PROGRAM SEQ_COSMO
VAR_INPUT
	COSMO_sequence	: UINT;
END_VAR

VAR
	process_V	: UINT; //COSMO to Pitstop
	process_W	: UINT; //COSMO to Reject Out
	process_X	: UINT; //Conveyor to Pitstop
	process_G	: UINT; //KR1 GET Magnet	
END_VAR


IF NOT AUTO_MODE.COSMO_LOAD OR GVL.KR1_EOAT_SUCTION OR GVL.LAYERPAD OR AUTO_MODE.FG_PACKING THEN
	RETURN;
END_IF

CASE COSMO_sequence OF
	0:
		process_V	:= 0;
		process_W	:= 0;
		process_X	:= 0;
		process_G	:= 0;
		COSMO_sequence := 1;		
		GVL.COSMO_UNLOAD := TRUE;
		AUTO_MODE.processnameCOSMO := CONCAT(MSG.COMP_CM,MSG.ACTION_INIT);
		LOGPROCESS( spLogComp	 := MSG.COMP_CM, 
		 			spLogAction	 := MSG.ACTION_INIT, 
		 			spLogStatus	 := MSG.STATUS_DONE,
	 	 		 	plogFlag	 := TRUE);
		
	// Get Magnet -------------------------------------------------------------------------------------------------------------	
	1:
		IF NOT GVL.KR1_EOAT_FILL AND NOT GVL.KR1_EOAT_SUCTION THEN
			IF process_G = 0 THEN
				IF KR1.Idle THEN
//					KR1.PLC_O_D3.0 := TRUE; //200
					KR1.bOutBit[3,0] := TRUE;
					AUTO_MODE.processnameCOSMO := CONCAT(MSG.COMP_CM,MSG.ACTION_GET_MAGNET);
					AUTO_MODE.processnameCOSMO := CONCAT(AUTO_MODE.processnameCOSMO,MSG.STATUS_RUN);
					LOGPROCESS( spLogComp	 := MSG.COMP_CM, 
								spLogAction	 := MSG.ACTION_GET_MAGNET, 
								spLogStatus	 := MSG.STATUS_RUN,
								plogFlag	 := TRUE);
					process_G := 1;
					RETURN;
				END_IF
			ELSIF process_G = 1 THEN
//				KR1.PLC_O_D3.0 := TRUE; //200
				KR1.bOutBit[3,0] := TRUE;
				IF NOT KR1.bInBit[3,0] THEN
//					KR1.PLC_O_D3.0 := FALSE; //200	
					KR1.bOutBit[3,0] := FALSE;
					AUTO_MODE.processnameCOSMO := CONCAT(MSG.COMP_CM,MSG.ACTION_GET_MAGNET);
					AUTO_MODE.processnameCOSMO := CONCAT(AUTO_MODE.processnameCOSMO,MSG.STATUS_ACK);
					LOGPROCESS( spLogComp	 := MSG.COMP_CM, 
								spLogAction	 := MSG.ACTION_GET_MAGNET, 
								spLogStatus	 := MSG.STATUS_ACK,
								plogFlag	 := TRUE);
					process_G := 2;
					RETURN;
				END_IF	
			ELSIF process_G = 2 THEN
//				KR1.PLC_O_D3.0 := FALSE; //200
				KR1.bOutBit[3,0] := FALSE;	
				IF KR1.bInBit[3,0] THEN
					AUTO_MODE.processnameCOSMO := CONCAT(MSG.COMP_CM,MSG.ACTION_GET_MAGNET);
					AUTO_MODE.processnameCOSMO := CONCAT(AUTO_MODE.processnameCOSMO,MSG.STATUS_DONE);
					LOGPROCESS( spLogComp	 := MSG.COMP_CM, 
								spLogAction	 := MSG.ACTION_GET_MAGNET, 
								spLogStatus	 := MSG.STATUS_DONE,
								plogFlag	 := TRUE);
					process_G:= 3;
					RETURN;
				END_IF	
			ELSIF process_G = 3 THEN
				IF KR1.Idle THEN
					AUTO_MODE.processnameCOSMO := CONCAT(MSG.COMP_CM,MSG.ACTION_GET_MAGNET);
					AUTO_MODE.processnameCOSMO := CONCAT(AUTO_MODE.processnameCOSMO,MSG.STATUS_COMP);
					LOGPROCESS( spLogComp	 := MSG.COMP_CM, 
								spLogAction	 := MSG.ACTION_GET_MAGNET, 
								spLogStatus	 := MSG.STATUS_COMP,
								plogFlag	 := TRUE);
					process_G := 4;
					COSMO_sequence := 2;
					AUTO_MODE.next_step := FALSE;
					GVL.KR1_EOAT_FILL := TRUE;
				END_IF
			END_IF
		ELSE
			COSMO_sequence := 2;
		END_IF
		
	// COSMO test --------------------------------------------------------------------------------------------------------------		
	2: 
		IF GVL.COSMO_OK THEN
			GVL.COSMO_Run := FALSE;
			AUTO_MODE.COSMO_RUN := FALSE;
			AUTO_MODE.processnameCOSMO := CONCAT(MSG.COMP_CM,MSG.ACTION_COSMO_PASS);
			AUTO_MODE.processnameCOSMO := CONCAT(AUTO_MODE.processnameCOSMO,MSG.STATUS_DONE);
			LOGPROCESS( spLogComp	 := MSG.COMP_CM, 
						spLogAction	 := MSG.ACTION_COSMO_PASS, 
						spLogStatus	 := MSG.STATUS_DONE,
						plogFlag	 := TRUE);
			COSMO_sequence := 3;
			AUTO_MODE.next_step := FALSE;
			AUTO_MODE.CLEAR_COSMO := TRUE;
			RETURN;
		ELSIF GVL.COSMO_NOTOK THEN
			GVL.COSMO_Run := FALSE;
			AUTO_MODE.COSMO_RUN := FALSE;
			AUTO_MODE.processnameCOSMO := CONCAT(MSG.COMP_CM,MSG.ACTION_COSMO_FAIL);
			AUTO_MODE.processnameCOSMO := CONCAT(AUTO_MODE.processnameCOSMO,MSG.STATUS_DONE);
			LOGPROCESS( spLogComp	 := MSG.COMP_CM, 
						spLogAction	 := MSG.ACTION_COSMO_FAIL, 
						spLogStatus	 := MSG.STATUS_DONE,
						plogFlag	 := TRUE);
			COSMO_sequence := 3;
			AUTO_MODE.next_step := FALSE;
			AUTO_MODE.CLEAR_COSMO := TRUE;
			RETURN;
		END_IF
			
	// COSMO to Reject Out -------------------------------------------------------------------------------------------------------------	
	3: 
			IF process_W = 0 THEN
				IF NOT AUTO_MODE.KR1_PITSTOP AND KR1.Idle AND NOT GVL.Conveyor_Full AND GVL.KR1_EOAT_FILL AND NOT AUTO_MODE.FG_PACKING AND NOT AUTO_MODE.RW_PACKING THEN
					KR1.bOutBit[3,6] := TRUE; //206
					AUTO_MODE.processnameCOSMO := CONCAT(MSG.COMP_CM,MSG.ACTION_COSMO_TO_CNVYR);
					AUTO_MODE.processnameCOSMO := CONCAT(AUTO_MODE.processnameCOSMO,MSG.STATUS_RUN);
					LOGPROCESS( spLogComp	 := MSG.COMP_CM, 
								spLogAction	 := MSG.ACTION_COSMO_TO_CNVYR, 
								spLogStatus	 := MSG.STATUS_RUN,
								plogFlag	 := TRUE);
					process_W := 1;
					RETURN;
				END_IF
			ELSIF process_W = 1 THEN
				KR1.bOutBit[3,6]:= TRUE; //206
				IF KR1.bInBit[3,6] THEN
					KR1.bOutBit[3,6] := FALSE; //2056
					AUTO_MODE.processnameCOSMO := CONCAT(MSG.COMP_CM,MSG.ACTION_COSMO_TO_CNVYR);
					AUTO_MODE.processnameCOSMO := CONCAT(AUTO_MODE.processnameCOSMO,MSG.STATUS_ACK);
					LOGPROCESS( spLogComp	 := MSG.COMP_CM, 
								spLogAction	 := MSG.ACTION_COSMO_TO_CNVYR, 
								spLogStatus	 := MSG.STATUS_ACK,
								plogFlag	 := TRUE);
					process_W := 2;
					RETURN;
				END_IF	
			ELSIF process_W = 2 THEN
				KR1.bOutBit[3,6] := FALSE; //206
				IF NOT KR1.bInBit[3,6] THEN
					AUTO_MODE.processnameCOSMO := CONCAT(MSG.COMP_CM,MSG.ACTION_COSMO_TO_CNVYR);
					AUTO_MODE.processnameCOSMO := CONCAT(AUTO_MODE.processnameCOSMO,MSG.STATUS_DONE);
					LOGPROCESS( spLogComp	 := MSG.COMP_CM, 
								spLogAction	 := MSG.ACTION_COSMO_TO_CNVYR, 
								spLogStatus	 := MSG.STATUS_DONE,
								plogFlag	 := TRUE);
					process_W:= 3;
					RETURN;
				END_IF
			ELSIF process_W = 3 THEN
				IF KR1.Idle THEN
						AUTO_MODE.processnameCOSMO := CONCAT(MSG.COMP_CM,MSG.ACTION_COSMO_TO_CNVYR);
						AUTO_MODE.processnameCOSMO := CONCAT(AUTO_MODE.processnameCOSMO,MSG.STATUS_COMP);
						LOGPROCESS( spLogComp	 := MSG.COMP_CM, 
									spLogAction	 := MSG.ACTION_COSMO_TO_CNVYR, 
									spLogStatus	 := MSG.STATUS_COMP,
									plogFlag	 := TRUE);
						process_W := 4;
						COSMO_sequence := 4;
						AUTO_MODE.next_step := FALSE;
						AUTO_MODE.CR_UNLOADING := FALSE;
						AUTO_MODE.CLEAR_COSMO := FALSE;
						GVL.Fail_Counter := GVL.Fail_Counter+1;
					END_IF
			END_IF	
	
	4:
		COSMO_sequence := 0;
		AUTO_MODE.next_step := FALSE;
		AUTO_MODE.COSMO_LOAD := FALSE;
		AUTO_MODE.CR_UNLOADING := FALSE;
		AUTO_MODE.CLEAR_COSMO := FALSE;
		GVL.COSMO_UNLOAD := FALSE;
		AUTO_MODE.processnameCOSMO := CONCAT(MSG.COMP_CM,MAIN.fb_TimeStamp.SystemTime);
		AUTO_MODE.processnameCOSMO := CONCAT(AUTO_MODE.processnameCOSMO,MSG.STATUS_END);
		AUTO_MODE.processnameCOSMO := CONCAT(MSG.COMP_CM,MSG.ACTION_COSMO);
		AUTO_MODE.processnameCOSMO := CONCAT(AUTO_MODE.processnameCOSMO,MSG.STATUS_END);
		LOGPROCESS( spLogComp	 := MSG.COMP_CM, 
					spLogAction	 := MSG.ACTION_COSMO, 
					spLogStatus	 := MSG.STATUS_END,
					plogFlag	 := TRUE);
END_CASE

END_PROGRAM

(* stored: Version 1.1.0.1, ProductVersion 3.1.4024.12
   POU SEQ_COSMO: Id {c67e620b-5c40-4e9a-8efa-f159aa47c021}, SpecialFunc None *)
